{attribute addProperty BoxType "EK1100-0000-0018"}
{attribute addProperty Id "A_0018_BK1250_0000_0019A_0018_BK1250_0000_0019_5BA9B27C00"}
{attribute addProperty CRC "3981104877"}
{attribute addProperty SizeInBites "0"}
{attribute addProperty SizeInBytes "0"}
TYPE Term_476_EK1100_ED4AD6ED EXTENDS EK1100_179A0949 :
STRUCT
	{attribute addProperty Name "A_0018_BK1250_0000_0019"}
	A_0018_BK1250_0000_0019 : A_0018_BK1250_0000_0019_5BA9B27C;
END_STRUCT
END_TYPE

(* stored: Version 1.2.0.0, ProductVersion 3.1.4024.9
   DUT Term_476_EK1100_ED4AD6ED: Id {4a223843-8657-4f97-9fb4-640c6db4cf48} *)
